{attribute addProperty BoxType "EL1502-0000-0018"}
{attribute addProperty Id "StatusAT %I*Status_20E8A7611621Counter_valueAT %I*UDINT32417"}
{attribute addProperty CRC "2441036875"}
{attribute addProperty SizeInBites "48"}
{attribute addProperty SizeInBytes "6"}
TYPE CNT_Inputs_917F444B :
STRUCT
	{attribute addProperty Name "Status"}
	Status AT %I* : Status_20E8A761;
	{attribute addProperty Name "Counter_value"}
	Counter_value AT %I* : UDINT;
END_STRUCT
END_TYPE

(* stored: Version 1.2.0.0, ProductVersion 3.1.4024.9
   DUT CNT_Inputs_917F444B: Id {2437fd01-27c7-441f-bf39-f842e85ba2a3} *)
